{attribute 'GeneratedUsingTerminal: AT2020-0250-0023'}
{attribute addProperty BoxType "AT2020-0250-0023"}
{attribute addProperty Id "A_0073_AT2000_5250_0016_AT2000_5250AT2000_01D6DEDF80"}
{attribute addProperty CRC "3204798256"}
{attribute addProperty Size "80"}
TYPE A_0061_AT2020_0250_0023_AT2020_0250_BF055730 EXTENDS AT2020_86175B41 :
STRUCT
	{attribute addProperty Name "A_0073_AT2000_5250_0016_AT2000_5250"}
	A_0073_AT2000_5250_0016_AT2000_5250 : AT2000_01D6DEDF;
END_STRUCT
END_TYPE

(* stored: Version 1.2.0.0, ProductVersion 3.1.4024.9
   DUT A_0061_AT2020_0250_0023_AT2020_0250_BF055730: Id {db00a32c-18a9-41f0-8cd4-8531d808208c} *)
